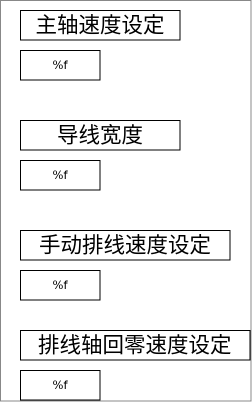
VISUALIZATION HMI1  // 252x402
    Rectangle (20,10 160x30), "主轴速度设定"
    Rectangle (20,50 80x30), "%f", text variable: MAIN.TargetMainAxisSpeed
        OnMouseDown: write the text variable via VisuDialogs.Numpad, min 0, max 20
    Rectangle (20,120 160x30), "导线宽度"
    Rectangle (20,230 210x30), "手动排线速度设定"
    Rectangle (20,330 230x30), "排线轴回零速度设定"
    Rectangle (20,160 80x30), "%f", text variable: MAIN.WireWeights
        OnMouseDown: write the text variable via VisuDialogs.Numpad, min 0, max 5
    Rectangle (20,270 80x30), "%f", text variable: MAIN.ManualControlVelocity
        OnMouseDown: write the text variable via VisuDialogs.Numpad, min 0, max 10
    Rectangle (20,370 80x30), "%f", text variable: MAIN.SlaveAxisBackZero
        OnMouseDown: write the text variable via VisuDialogs.Numpad, min 0, max 10
END_VISUALIZATION

(* stored: Version 1.1.0.1, ProductVersion 3.1.4024.12
   Visu HMI1: Id {0a0ea37a-475d-476a-b0e5-f9b1924c58d4} *)
